PROGRAM MAIN
VAR
	Machine : FB_Machine;
END_VAR

Machine(
	Ctrl:= GVL_Remote.Ctrl, 
	Status:= GVL_Remote.Status, 
	Service:= GVL_Remote.Service, 
	Admin:= GVL_Remote.Admin);

END_PROGRAM

(* stored: Version 1.1.0.1, ProductVersion 3.1.4026.18
   POU MAIN: Id {ff2cc2b3-37fa-4751-9ea9-2181601b74ac}, SpecialFunc None *)
